FUNCTION_BLOCK FB_FanControl
VAR_INPUT
	fSpeed	:	REAL;		//Fan speed setpoint 0..100%
END_VAR
VAR
	fSpeedSetRaw  AT%Q*	: REAL 	:=0; 	//Raw value for terminal => send to valve
END_VAR
VAR CONSTANT
		fFactor : REAL :=327.67;	// factor for calculating the terminal integer values (from percentage to int)
END_VAR

fSpeedSetRaw := fSpeed;

END_FUNCTION_BLOCK

(* stored: Version 1.1.0.1, ProductVersion 3.1.4024.9
   POU FB_FanControl: Id {643c59a2-f668-40c9-a3c5-9486aaf77939}, SpecialFunc None *)
